FUNCTION_BLOCK L2_MachineINIT (* Basic Function Block Type *)
  (* Standard: 61499-2 *)
  (* Version 0.0, 2016-01-15, EQUEROL, UJI *)
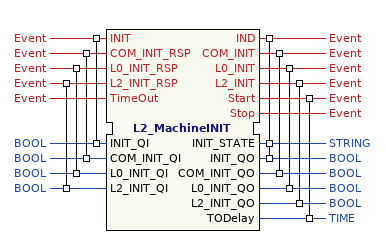
  EVENT_INPUT
    INIT WITH INIT_QI; (* Initialization Request *)
    COM_INIT_RSP WITH COM_INIT_QI; (* Communication initialization response *)
    L0_INIT_RSP WITH L0_INIT_QI; (* Respone to the initialization request sent to L0 *)
    L2_INIT_RSP WITH L2_INIT_QI; (* Layer 2 blocks initialization response *)
    TimeOut; (* Initialization timeout *)
  END_EVENT
  EVENT_OUTPUT
    IND WITH INIT_STATE, INIT_QO; (* Indicate initialization result *)
    COM_INIT WITH COM_INIT_QO; (* Initialize the communications FBs with L3,L1 and L0 *)
    L0_INIT WITH L0_INIT_QO; (* Initialization Confirm *)
    L2_INIT WITH L2_INIT_QO; (* Layer 2 blocks initialization request *)
    Start WITH TODelay; (* Start the delay to control initialization timeout *)
    Stop; (* Stop the delay to control initialization timeout *)
  END_EVENT
  VAR_INPUT
    INIT_QI : BOOL; (* Initialization qualifier *)
    COM_INIT_QI : BOOL; (* Comunications initialization qualifier *)
    L0_INIT_QI : BOOL; (* L0 initialization qualifier *)
    L2_INIT_QI : BOOL; (* Layer 2 initialization qualifier *)
  END_VAR
  VAR_OUTPUT
    INIT_STATE : STRING; (* String containing the state of the initialization *)
    INIT_QO : BOOL; (* Initialization output qualifier *)
    COM_INIT_QO : BOOL; (* Communication initialization qualifier *)
    L0_INIT_QO : BOOL; (* Output event qualifier *)
    L2_INIT_QO : BOOL; (* Layer 2 blocks initialization qualifier *)
    TODelay : TIME; (* Timeout delay *)
  END_VAR
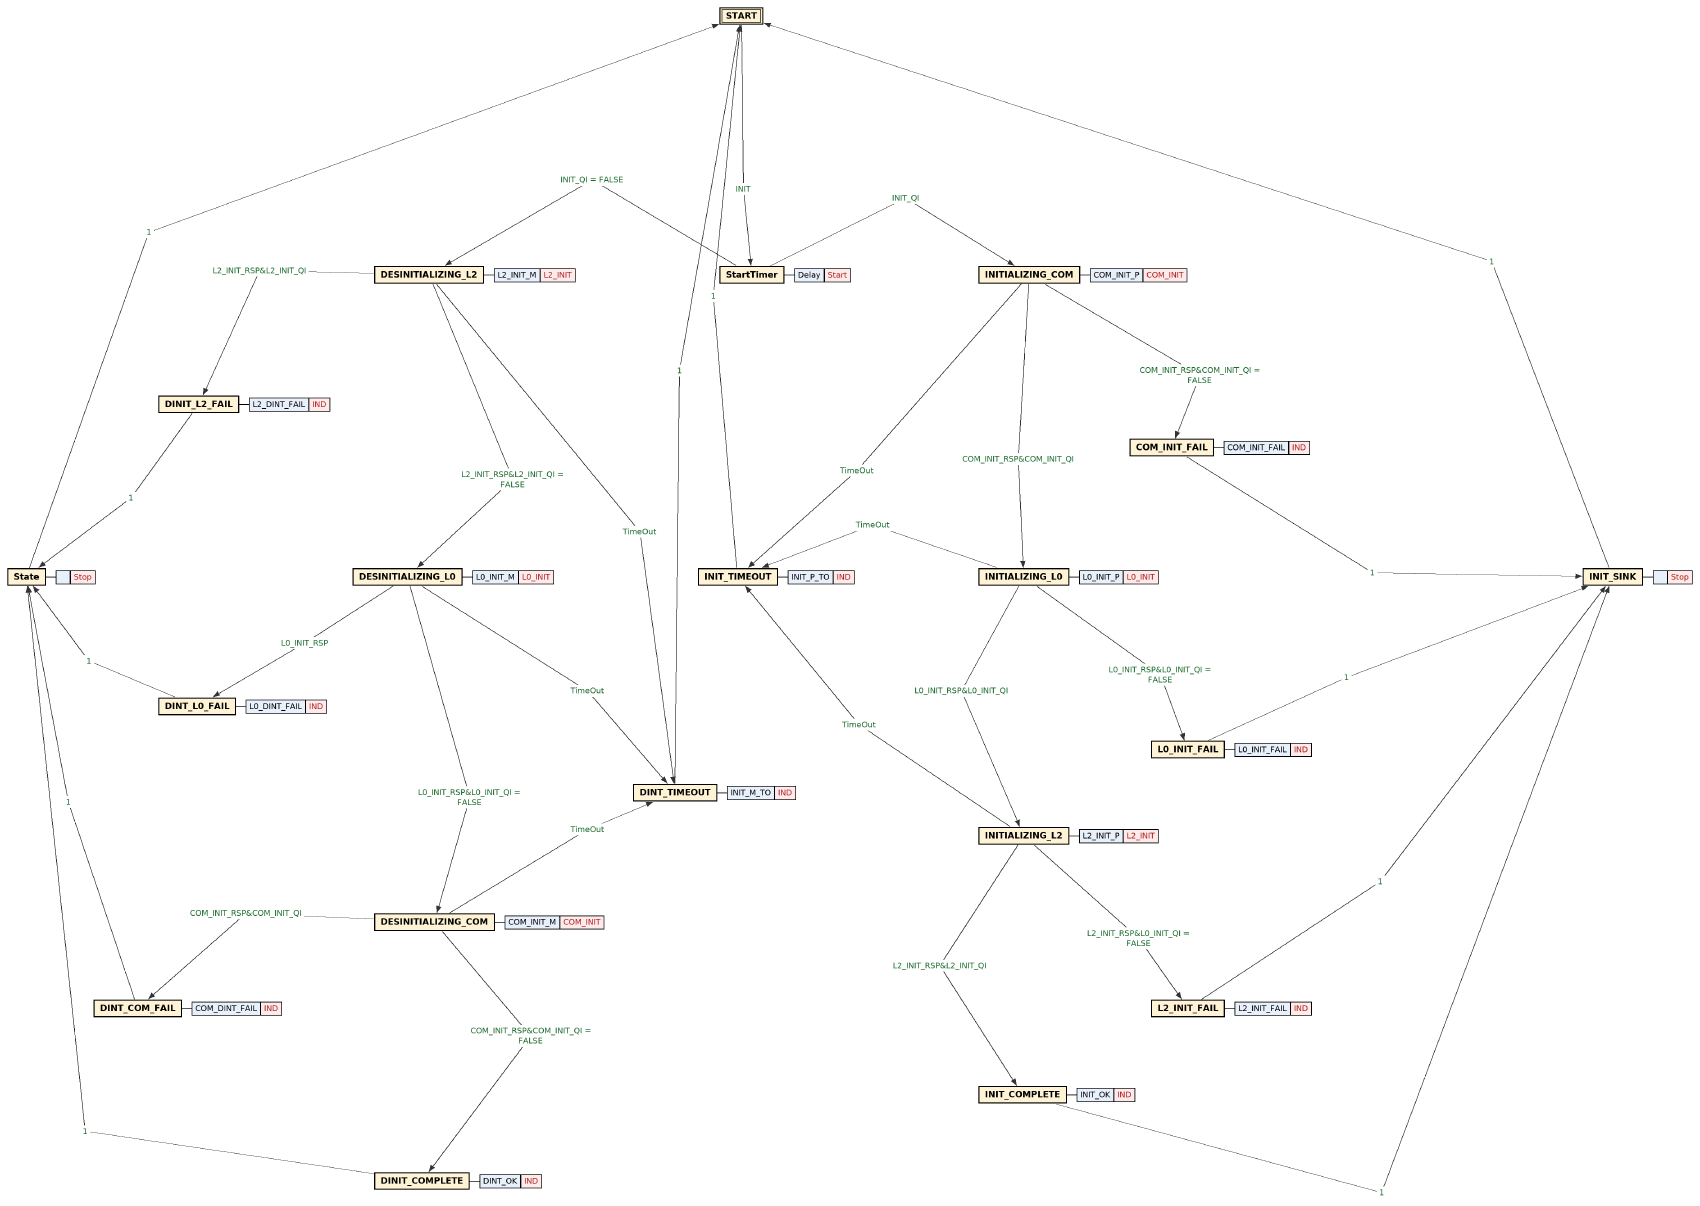
  EC_STATES
    START; (* Initial State *)
    INITIALIZING_COM : COM_INIT_P -> COM_INIT;
    DESINITIALIZING_L0 : L0_INIT_M -> L0_INIT;
    INIT_COMPLETE : INIT_OK -> IND;
    INIT_SINK : -> Stop;
    INITIALIZING_L0 : L0_INIT_P -> L0_INIT;
    COM_INIT_FAIL : COM_INIT_FAIL -> IND;
    L0_INIT_FAIL : L0_INIT_FAIL -> IND;
    INITIALIZING_L2 : L2_INIT_P -> L2_INIT;
    L2_INIT_FAIL : L2_INIT_FAIL -> IND;
    DESINITIALIZING_COM : COM_INIT_M -> COM_INIT;
    DESINITIALIZING_L2 : L2_INIT_M -> L2_INIT;
    StartTimer : Delay -> Start;
    INIT_TIMEOUT : INIT_P_TO -> IND;
    DINIT_COMPLETE : DINT_OK -> IND;
    State : -> Stop;
    DINIT_L2_FAIL : L2_DINT_FAIL -> IND;
    DINT_L0_FAIL : L0_DINT_FAIL -> IND;
    DINT_COM_FAIL : COM_DINT_FAIL -> IND;
    DINT_TIMEOUT : INIT_M_TO -> IND;
  END_STATES
  EC_TRANSITIONS
    INITIALIZING_COM TO INITIALIZING_L0 := COM_INIT_RSP&COM_INIT_QI;
    INITIALIZING_COM TO COM_INIT_FAIL := COM_INIT_RSP&COM_INIT_QI = FALSE;
    COM_INIT_FAIL TO INIT_SINK := 1;
    L0_INIT_FAIL TO INIT_SINK := 1;
    INITIALIZING_L0 TO INITIALIZING_L2 := L0_INIT_RSP&L0_INIT_QI;
    INITIALIZING_L0 TO L0_INIT_FAIL := L0_INIT_RSP&L0_INIT_QI = FALSE;
    L2_INIT_FAIL TO INIT_SINK := 1;
    INITIALIZING_L2 TO L2_INIT_FAIL := L2_INIT_RSP&L0_INIT_QI = FALSE;
    INITIALIZING_L2 TO INIT_COMPLETE := L2_INIT_RSP&L2_INIT_QI;
    INIT_SINK TO START := 1;
    START TO StartTimer := INIT;
    StartTimer TO INITIALIZING_COM := INIT_QI;
    StartTimer TO DESINITIALIZING_L2 := INIT_QI = FALSE;
    INITIALIZING_COM TO INIT_TIMEOUT := TimeOut;
    INITIALIZING_L0 TO INIT_TIMEOUT := TimeOut;
    INITIALIZING_L2 TO INIT_TIMEOUT := TimeOut;
    INIT_COMPLETE TO INIT_SINK := 1;
    INIT_TIMEOUT TO START := 1;
    DESINITIALIZING_L2 TO DESINITIALIZING_L0 := L2_INIT_RSP&L2_INIT_QI = FALSE;
    DESINITIALIZING_L2 TO DINIT_L2_FAIL := L2_INIT_RSP&L2_INIT_QI;
    DINIT_L2_FAIL TO State := 1;
    DESINITIALIZING_L0 TO DESINITIALIZING_COM := L0_INIT_RSP&L0_INIT_QI = FALSE;
    DESINITIALIZING_L0 TO DINT_L0_FAIL := L0_INIT_RSP;
    DINT_L0_FAIL TO State := 1;
    DESINITIALIZING_COM TO DINIT_COMPLETE := COM_INIT_RSP&COM_INIT_QI = FALSE;
    DESINITIALIZING_COM TO DINT_COM_FAIL := COM_INIT_RSP&COM_INIT_QI;
    DINT_COM_FAIL TO State := 1;
    DINIT_COMPLETE TO State := 1;
    DESINITIALIZING_COM TO DINT_TIMEOUT := TimeOut;
    DESINITIALIZING_L0 TO DINT_TIMEOUT := TimeOut;
    DESINITIALIZING_L2 TO DINT_TIMEOUT := TimeOut;
    DINT_TIMEOUT TO START := 1;
    State TO START := 1;
  END_TRANSITIONS
  ALGORITHM COM_INIT_P IN ST: (* new algorithm *)
COM_INIT_QO := TRUE;
  END_ALGORITHM
  ALGORITHM COM_INIT_FAIL IN ST: (* new algorithm *)
INIT_STATE := "Unable to start communications with L3,L1 and L0";
INIT_QO := FALSE;
  END_ALGORITHM
  ALGORITHM L0_INIT_P IN ST: (* new algorithm *)
L0_INIT_QO := TRUE;
  END_ALGORITHM
  ALGORITHM L0_INIT_FAIL IN ST: (* new algorithm *)
INIT_STATE := "Unable to initialize L0 device";
INIT_QO := FALSE;
  END_ALGORITHM
  ALGORITHM L2_INIT_P IN ST: (* new algorithm *)
L2_INIT_QO := TRUE;
  END_ALGORITHM
  ALGORITHM L2_INIT_FAIL IN ST: (* new algorithm *)
INIT_STATE := "Unable to initialize machine own FBs";
INIT_QO := FALSE;
  END_ALGORITHM
  ALGORITHM INIT_OK IN ST: (* new algorithm *)
INIT_STATE := "Initialization OK";
INIT_QO := TRUE;
  END_ALGORITHM
  ALGORITHM Delay IN ST: (* new algorithm *)
TODelay := TIME#30s;
  END_ALGORITHM
  ALGORITHM INIT_P_TO IN ST: (* new algorithm *)
INIT_STATE := "Initialization timeout (30s timer expired)";
INIT_QO := FALSE;
  END_ALGORITHM
  ALGORITHM L2_INIT_M IN ST: (* new algorithm *)
L2_INIT_QO := FALSE;
  END_ALGORITHM
  ALGORITHM L2_DINT_FAIL IN ST: (* new algorithm *)
INIT_STATE := "Unable to stop machine own FBs";
INIT_QO := TRUE;
  END_ALGORITHM
  ALGORITHM L0_INIT_M IN ST: (* new algorithm *)
L0_INIT_QO := FALSE;
  END_ALGORITHM
  ALGORITHM L0_DINT_FAIL IN ST: (* new algorithm *)
INIT_STATE := "Unable to desinitialize L0 device";
INIT_QO := TRUE;
  END_ALGORITHM
  ALGORITHM COM_INIT_M IN ST: (* new algorithm *)
COM_INIT_QO := FALSE;
  END_ALGORITHM
  ALGORITHM COM_DINT_FAIL IN ST: (* new algorithm *)
INIT_STATE := "Unable to stop communications with L3,L1 and L0";
INIT_QO := TRUE;
  END_ALGORITHM
  ALGORITHM DINT_OK IN ST: (* new algorithm *)
INIT_STATE := "Desinitialization OK";
INIT_QO := FALSE;
  END_ALGORITHM
  ALGORITHM INIT_M_TO IN ST: (* new algorithm *)
INIT_STATE := "Desinitialization timeout (30s timer expired)";
INIT_QO := TRUE;
  END_ALGORITHM
END_FUNCTION_BLOCK
